FUNCTION_BLOCK GasolineMotor EXTENDS Motor

METHOD PUBLIC LoadFuel
ADSLOGSTR(    msgCtrlMask:=ADSLOG_MSGTYPE_LOG,
              msgFmtStr:='Loading fuel into the Gasoline motor..',
              strArg:='');
END_METHOD

METHOD PUBLIC SpeedUp
ADSLOGSTR(    msgCtrlMask:=ADSLOG_MSGTYPE_LOG,
              msgFmtStr:='Accelerating the Gasoline motor...',
              strArg:='');
END_METHOD

METHOD PUBLIC StartUp
ADSLOGSTR(    msgCtrlMask:=ADSLOG_MSGTYPE_LOG,
              msgFmtStr:='Starting the Gasoline motor...',
              strArg:='');
END_METHOD

METHOD PUBLIC Stop
ADSLOGSTR(    msgCtrlMask:=ADSLOG_MSGTYPE_LOG,
              msgFmtStr:='Stopping the Gasoline motor...',
              strArg:='');
END_METHOD

END_FUNCTION_BLOCK

(* stored: Version 1.1.0.1, ProductVersion 3.1.4024.12
   POU GasolineMotor: Id {2ddba2a9-c57d-4337-a725-f74b361c1c46}, SpecialFunc None
   Method LoadFuel: Id {496ded0f-2372-4bf9-adcd-44b0d2a3e619}
   Method SpeedUp: Id {fc2288e7-a842-4348-99e3-ef75ab71952a}
   Method StartUp: Id {78539401-4b6c-4b49-a534-9d7a54f66669}
   Method Stop: Id {d33a00f8-2969-4a17-9821-a289cbf74861} *)
